INTERFACE I_ContinuousDrive EXTENDS I_Drive

METHOD ABSTRACT moveContinuous : BOOL
VAR_INPUT
	newDirection : MC_Direction;
END_VAR
END_METHOD

END_INTERFACE

(* stored: Version 1.1.0.1, ProductVersion 3.1.4024.11
   Itf I_ContinuousDrive: Id {8029c368-6f74-418f-8fb7-9c63a351cb8c}
   Method moveContinuous: Id {f9f5760b-5ae9-4bfa-9e9a-44fb05051f3f} *)
